Staubli VAL3: WriteSingIOMsg.dtx

public Body body
  [0]
    num nData[9]
public Header header
  [0]
    num nCommType
    num nData[12]
    num nMsgType
    num nReplyCode
public Prefix prefix
  [0]
    num nData[4]
    num nLength
public WriteSingleIO writeSingleIO
  [0]
    bool bState
    num nModuleId
    num nPin
